(* IEC 61131-3 sources: SamplePLCprogramming/bbi_trendN (part 2) *)

(* ---- bbi_trendN.fun ---- *)
FUNCTION fFileFilter : BOOL
	VAR_INPUT
		filter : USINT;
		strlen : INT;
		pString : UDINT;
	END_VAR
	VAR
		i : INT;
		aChar : REFERENCE TO USINT;
		lastPoint : INT;
		aString : REFERENCE TO STRING[40];
	END_VAR
END_FUNCTION

FUNCTION_BLOCK fMakeTrendData
	VAR_INPUT
		ncCLthis : USINT;
		ncOthis : USINT;
		ncIthis : USINT;
		stack : trendStack_typ;
		time : DATE_AND_TIME;
		new : BOOL;
	END_VAR
	VAR_OUTPUT
		data : ARRAY[0..1023] OF USINT;
		dataLen : UDINT;
	END_VAR
	VAR
		dataLineTrend : batchf_max_data_typ;
		oldstack : trendStack_typ;
		CRC : REFERENCE TO UDINT;
		aUDINT : REFERENCE TO UDINT;
		aReal : REFERENCE TO REAL;
		aCRLF : REFERENCE TO ARRAY[0..3] OF USINT;
		count : USINT;
		i : USINT;
	END_VAR
END_FUNCTION_BLOCK

FUNCTION_BLOCK fTrendRead
	VAR_IN_OUT
		c : trendReadCtrl_typ;
		y : ARRAY[0..nTRENDCHANNELS] OF trend_read_channel_typ;
	END_VAR
	VAR
		cCLmax : USINT;
		cOmax : USINT;
		cImax : USINT;
		allChannelsMax : USINT; (*Anzahl!! aller kanäle in erster Datenzeile (Vollbelegung)*)
		allchannelsThisSample : USINT; (*Anzahl der Kanäle im neuen Sample*)
		curAge : REAL; (*batchage in der gerade geschriebene CSV Zeile*)
		DirCreate_0 : DirCreate;
		FileCreate_0 : FileCreate;
		FileOpen_0 : FileOpen;
		FileWriteEx_0 : FileWriteEx;
		FileClose_0 : FileClose;
		identCSV : UDINT;
		CRCB : UDINT;
		CRCA : UDINT;
		copyHeader : {REDUND_UNREPLICABLE} batchf_header_typ;
		aHead : REFERENCE TO batchf_header_typ;
		aDataA : REFERENCE TO batchf_max_dataA_typ;
		aCRC : REFERENCE TO UDINT;
		aReal : REFERENCE TO REAL;
		hlpstr2 : STRING[5];
		hlpstr : STRING[100];
		dataDel : ARRAY[0..3] OF USINT := [DATA_LINE_STARTCHAR1,DATA_LINE_STARTCHAR2,DATA_LINE_STARTCHAR3,DATA_LINE_STARTCHAR4]; (*Datenpaket Markierung*)
		targetTimeOffsetMsec : UDINT; (*Msec Übertrag aus letztem Plotting als Offset für nächtes Plotten*)
		targetTimeIncMsec : UDINT; (*Increment für Zielzeit in Msec*)
		targetTimeSecAbs : UDINT; (*!!absolute!! Zielzeit in Sekunden für Trendobjekt Sample*)
		dT : UDINT; (*Rohsample Zeitdifferen in Msec*)
		tx : UDINT; (*Interpolationspunkt in Msec zwischen den Rohsamples*)
		bufReadTrend : UDINT; (*fertig verarbeitete bytes im aktuellen Trend Puffer Block*)
		buflenCSV : UDINT; (*fertig aufbereitet bytes im CSV Schreibpuffer*)
		lastV : ARRAY[0..ALLCHANNELS] OF REAL; (*letzte entpackte Datenzeile *)
		curV : ARRAY[0..ALLCHANNELS] OF REAL; (*aktuell entpackte Datenzeile *)
		bufCSV : ARRAY[0..CSV_W_BUFSIZE] OF USINT; (*Schreibepuffer für CSV Datei*)
		skip : BOOL;
		lastT : UDINT;
		curT : UDINT;
		dY : ARRAY[0..nTRENDCHANNELS] OF REAL;
		Y2 : ARRAY[0..nTRENDCHANNELS] OF REAL;
		Y1 : ARRAY[0..nTRENDCHANNELS] OF REAL;
		i : USINT;
	END_VAR
	VAR CONSTANT
		SEMI : USINT := 59;
		CRLF : ARRAY[0..1] OF USINT := [13,10];
	END_VAR
	VAR
		timeGapRawSamples : UDINT; (*workaround zur ausreißererkennung*)
		indexOffset : USINT;
		STEP : USINT;
		offsetCSVFile : UDINT; (*Offset in der Augabedatei für Blockweises schreiben*)
		offsetTrendFile : UDINT;
		draw : BOOL;
	END_VAR
END_FUNCTION_BLOCK

FUNCTION_BLOCK fTrendWrite
	VAR_INPUT
		time : DATE_AND_TIME;
		freeMem : UDINT;
		filename : STRING[40]; (*Dateiname*)
		indexUnit : USINT;
		pATbuf : UDINT;
		pNon : UDINT;
		pRem : UDINT;
		enable : BOOL;
	END_VAR
	VAR_IN_OUT
		c : trendWriteCtrl_typ;
	END_VAR
	VAR
		lastFullSample : UDINT;
		hlpstr : STRING[100];
		aDel : REFERENCE TO ARRAY[0..3] OF USINT;
		bufoff : ARRAY[0..BATCH_OFFSETSEARCH] OF USINT;
		bufh_event_out : eventRecordHeader_typ;
		bufh_event_in : eventRecordHeader_typ;
		bufh_out : batchf_header_typ;
		bufh_in : batchf_header_typ;
		difOffset : UDINT;
		i : UDINT;
		gotOffset : BOOL;
		FileCreate_0 : FileCreate;
		FileClose_0 : FileClose;
		fMakeEventData_0 : fMakeEventData;
		fMakeTrendData_0 : fMakeTrendData;
		FileWrite_0 : FileWrite;
		debug1 : UDINT;
		FileReadEx_0 : FileReadEx;
	END_VAR
	VAR
		DirCreate_0 : DirCreate;
		FileOpen_0 : FileOpen;
		fileIdentEvent : UDINT;
		fileIdent : UDINT;
		fileOpenLenEvent : UDINT;
		fileOpenLen : UDINT;
		aNon : REFERENCE TO core_non_typ;
		aRem : REFERENCE TO config_rem_typ;
		countCloseRaw : USINT;
		countOpenRaw : USINT;
		STEP : USINT;
		stack : statusStack;
		ebuf : REFERENCE TO trail_buffer_typ;
		lastPop : UDINT;
		eventsToPop : UINT;
		e : trail_buffer_entry_typ;
		debug : USINT;
	END_VAR
END_FUNCTION_BLOCK

(* ---- Constants.var ---- *)
VAR CONSTANT
	BAT_W_STP_init : USINT := 0;
	BAT_R_STP_wait : USINT := 0;
	BAT_R_STA_waiting : USINT := 0; (*warte auf befehl, wenn alter befehl mit 0 quittiert wurde: ERFOLG*)
	BATCH_STARTED : USINT := 0;
	BAT_D_STA_waiting : USINT := 0;
	BAT_D_STP_wait : USINT := 0;
	BAT_W_STA_waiting : USINT := 0;
	BAT_D_STP_getInfo : USINT := 1;
	BAT_W_STA_initializing : USINT := 1;
	BAT_W_STP_open : USINT := 1;
	BAT_D_STA_gettingInfo : USINT := 1;
	BAT_W_STP_create : USINT := 2;
	BAT_R_STP_createDir : USINT := 2;
	BAT_D_STA_reading : USINT := 2;
	BAT_D_STP_read : USINT := 2;
	BAT_W_STA_recording : USINT := 2;
	BAT_W_STP_read_header : USINT := 3;
	BAT_D_STP_error : USINT := 3;
	BAT_D_STA_error : USINT := 3;
	BAT_R_STP_createCSV : USINT := 3;
	BAT_W_STA_starting : USINT := 3;
	BAT_R_STA_preparing : USINT := 3; (*einmalige Header checks der Rohdaten und Anlegen der CSV Kopfzeilen*)
	BAT_R_STA_unzipping : USINT := 4; (*Entpacke Daten*)
	BAT_R_STP_readData : USINT := 4;
	BAT_W_STA_stopping : USINT := 4;
	BAT_W_STP_write_header : USINT := 4;
	BAT_R_STA_newCSVfile : USINT := 5; (*alte CSV Datei schließen, neue CSV Datei öffnen*)
	BAT_R_STP_CSVfullHeader : USINT := 5;
	BAT_W_STP_write_data : USINT := 6;
	BAT_R_STP_CSVsmallHeader : USINT := 6;
	BAT_R_STA_closing : USINT := 7; (*CSC Datei Schließen und Status OK*)
	BAT_W_STP_get_offset : USINT := 7;
	BAT_R_STA_closingError : USINT := 8; (*CSC Datei Schließen nach Status Fehler*)
	BAT_R_STP_unzipCheck : USINT := 8;
	BAT_R_STA_closingAbort : USINT := 9; (*CSC Datei Schließen nach Abbruchbefehl*)
	BAT_D_LISTSLOTS : USINT := 9;
	BAT_R_STP_unzip : USINT := 9;
	BAT_R_CMD_trend : USINT := 10;
	BAT_R_STP_writeCSV : USINT := 10;
	BAT_W_STP_wait : USINT := 10;
	BAT_W_CMD_start : USINT := 10;
	BAT_R_STP_closeCSV : USINT := 12;
	BAT_W_CMD_stop : USINT := 20;
	BAT_R_CMD_csvFull : USINT := 20;
	BAT_W_STP_close : USINT := 20;
	BAT_W_STP_closeRec : USINT := 21;
	BAT_W_STP_dir : USINT := 22;
	BAT_R_CMD_csvSmall : USINT := 30;
	DATA_LINE_STARTCHAR2 : USINT := 35;
	DATA_LINE_STARTCHAR5 : USINT := 35;
	DATA_LINE_STARTCHAR4 : USINT := 36;
	DATA_LINE_STARTCHAR3 : USINT := 37;
	DATA_LINE_STARTCHAR1 : USINT := 38;
	DATA_LINE_ENDCHAR : USINT := 47;
	EVENT_W_STP_open : USINT := 51;
	EVENT_W_STP_dir : USINT := 52;
	EVENT_W_STP_create : USINT := 53;
	EVENT_W_STP_write_first : USINT := 54;
	EVENT_W_STP_write_header : USINT := 55;
	EVENT_W_STP_closeRec : USINT := 56;
	EVENT_W_STP_read_header : USINT := 57;
	EVENT_W_STP_get_offset : USINT := 58;
	EVENT_W_STP_error : USINT := 59;
	EVENT_W_STP_write_data : USINT := 60;
	EVENT_W_STP_close : USINT := 61;
	BAT_R_CMD_abort : USINT := 90;
	BAT_R_STA_error : USINT := 99; (*Fehler, siehe error struct*)
	BAT_W_STA_error : USINT := 99;
	BAT_W_STP_error : USINT := 99;
	BAT_R_STP_error : USINT := 99;
	BATCH_FINALIZED : USINT := 255;
	TRENDITEMS : UINT := 719; (*Anzahl der Bildpunkte / CSV - Datenzeilen*)
	BATCH_OFFSETSEARCH : UDINT := 1000;
	MAX_CHAR_CSV_ROW : UDINT := 4000; (*Maximalanzahl an Zeichen für entpackte Datenzeile die noch im CSV Schreibpuffer frei sein muss*)
	MAX_LINES_CSV : UDINT := 30000; (*Maximalanzahl an CSV Zeilen*)
	BAT_R_BUFSIZE : UDINT := 51200; (*Größe des Lesepuffers für Rohdaten*)
	CSV_W_BUFSIZE : UDINT := 51200; (*Größe des CSV Schreibpuffers*)
	TRENDPARTSIZE : UDINT := 31457280; (*Größe der DRAM Partition für Trend-Rohdatenabbild, 30 MB*)
	BATCH_GENERATOR : UDINT := 548942248;
	BAT_D_VIEWSLOTS : UDINT := BAT_D_LISTSLOTS+1;
END_VAR
(**)
